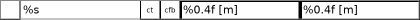
VISUALIZATION _VISU_CameraBaseSetting  // 420x20
VAR_IN_OUT
	m_Inst : FB_CameraBase;
END_VAR
    Rectangle (300,0 120x20), "%0.4f [m]", tooltip "CameraToPrintUnit", text variable: m_Inst._fCameraToPrintOffset
        OnMouseDown: write the text variable via Default
    Rectangle (180,0 120x20), "%0.4f [m]", tooltip "DetectToCamera", text variable: m_Inst._fDetectToCameraOffset
        OnMouseDown: write the text variable via Default
    RoundedRectangle (140,0 20x20), "ct", tooltip "UseCameraTrigger", colour toggle: m_Inst._bUseCameraTrigger
    RoundedRectangle (160,0 20x20), "cfb", tooltip "UseCameraTriggerFeedback", colour toggle: m_Inst._bUseCameraTriggerFeedback
    Rectangle (20,0 120x20), "%s", text variable: m_Inst.sName
    RoundedRectangle (0,0 20x20), tooltip "Camera activated", colour toggle: m_Inst._bActivated <> 0
END_VISUALIZATION

(* stored: Version 1.1.0.1, ProductVersion 3.1.4024.3
   Visu _VISU_CameraBaseSetting: Id {9f91569e-5850-41c5-8c2a-6e99eea6673b} *)
